(* Logix 5000 project; controller IPG_2332_07A 1769-L16ER-BB1B rev 34.12; software revision 34.01; part 2 of 4 *)
(* tags used below, declared in another part *)
   Axis_Controller : udt_Zaber_Axis;
   p_ALMD_00 : ALARM_DIGITAL;
   p_ALMD_01 : ALARM_DIGITAL;
   p_ALMD_02 : ALARM_DIGITAL;
   p_ALMD_03 : ALARM_DIGITAL;
   p_ALMD_04 : ALARM_DIGITAL;
   p_ALMD_05 : ALARM_DIGITAL;
   p_AOI_PLC_Status : AOI_PLC_Status;
   p_BarcodeDone : BOOL;
   p_CassetteGripper_Ext_IN : BOOL;
   p_CassetteGripper_OUT : BOOL;
   p_CassetteGripper_Ret_IN : BOOL;
   p_CassettePresence_IN : BOOL;
   p_CassetteRelease_IN : BOOL;   // Foot Switch
   p_Control : udt_Machine_Control_V2;   // Main Control
   p_DispenseStart_OUT : BOOL;
   p_DoorMonitor_IN : BOOL;
   p_EstopMonitor_IN : BOOL;
   p_EStopPB_IN : BOOL;
   p_EstopReset_OUT : BOOL;
   p_FerruleGripper_IN : BOOL;
   p_FerruleGripper_OUT : BOOL;
   p_FiberAxis : udt_Zaber_Axis;
   p_FiberAxis_FindPos : udt_Station_Sequence;
   p_FiberGripper_IN : BOOL;
   p_FiberGripper_OUT : BOOL;
   p_HMI_IO_Display : udt_HMI_IO_Desc;
   p_HMI_Message_Active : udt_HMI_Message_Display;
   p_HMI_Message_Sequence_Active : udt_HMI_Message_Display;
   p_HMI_PLC_Status : udt_Controller_Status;
   p_LED_01 : udt_LED;
   p_LED_02 : udt_LED;
   p_LED_03 : udt_LED;
   p_LED_04 : udt_LED;
   p_LED_Ramp_Done : BOOL;
   p_Machine_Control : udt_Machine_Control_V2;
   p_MainAirOkay_IN : BOOL;
   p_MirrorAxis : udt_Zaber_Axis;
   p_OkayToProcess : BOOL;
   p_PBLight_Amber_OUT : BOOL;
   p_PBLight_Green_OUT : BOOL;
   p_PBLight_Red_OUT : BOOL;
   p_Sequence : udt_Station_Sequence;
   p_StackLight_Amber_OUT : BOOL;
   p_StackLight_Green_OUT : BOOL;
   p_StackLight_Red_OUT : BOOL;
   p_StartPB_IN : BOOL;
   p_SyringeAxis : udt_Zaber_Axis;
   p_test_Mode : BOOL;
   p_Waiting : BOOL;
   p_WorkLight_OUT : BOOL;
   DateTime : DateTime;
   Debug_SDF : DINT;
   HMI_IO_Description : udt_IO_Desc[96];
   HMI_Messages : udt_HMI_Message_Display[48];
   HMI_Messages_Sequence : udt_HMI_Message_Display[20];
(* MainProgram_10Ms, continued *)

ROUTINE C_Alarm   (* ladder *)
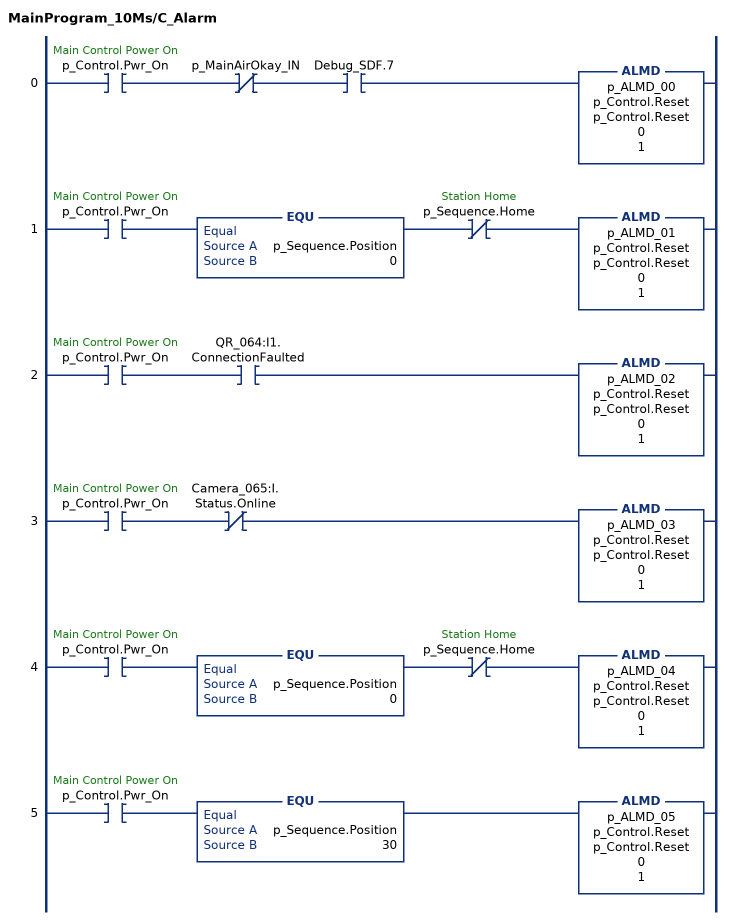
   0: XIC(p_Control.Pwr_On)XIO(p_MainAirOkay_IN)XIC(Debug_SDF.7)ALMD(p_ALMD_00,p_Control.Reset,p_Control.Reset,0,1);
   1: XIC(p_Control.Pwr_On)EQU(p_Sequence.Position,0)XIO(p_Sequence.Home)ALMD(p_ALMD_01,p_Control.Reset,p_Control.Reset,0,1);
   2: XIC(p_Control.Pwr_On)XIC(QR_064:I1.ConnectionFaulted)ALMD(p_ALMD_02,p_Control.Reset,p_Control.Reset,0,1);
   3: XIC(p_Control.Pwr_On)XIO(Camera_065:I.Status.Online)ALMD(p_ALMD_03,p_Control.Reset,p_Control.Reset,0,1);
   4: XIC(p_Control.Pwr_On)EQU(p_Sequence.Position,0)XIO(p_Sequence.Home)ALMD(p_ALMD_04,p_Control.Reset,p_Control.Reset,0,1);
   5: XIC(p_Control.Pwr_On)EQU(p_Sequence.Position,30)ALMD(p_ALMD_05,p_Control.Reset,p_Control.Reset,0,1);
END_ROUTINE

ROUTINE D_InputMapping   (* ladder *)
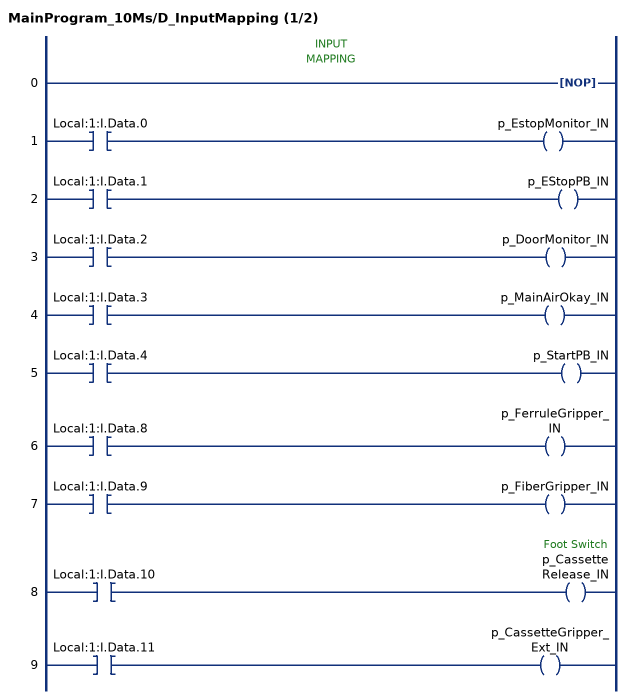
   // INPUT
   // MAPPING
   0: NOP();
   1: XIC(Local:1:I.Data.0)OTE(p_EstopMonitor_IN);
   2: XIC(Local:1:I.Data.1)OTE(p_EStopPB_IN);
   3: XIC(Local:1:I.Data.2)OTE(p_DoorMonitor_IN);
   4: XIC(Local:1:I.Data.3)OTE(p_MainAirOkay_IN);
   5: XIC(Local:1:I.Data.4)OTE(p_StartPB_IN);
   6: XIC(Local:1:I.Data.8)OTE(p_FerruleGripper_IN);
   7: XIC(Local:1:I.Data.9)OTE(p_FiberGripper_IN);
   8: XIC(Local:1:I.Data.10)OTE(p_CassetteRelease_IN);
   9: XIC(Local:1:I.Data.11)OTE(p_CassetteGripper_Ext_IN);
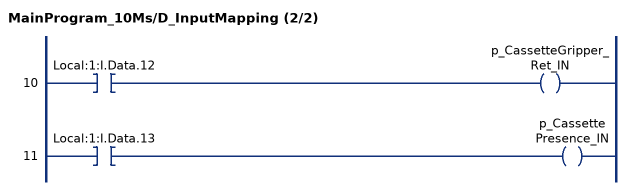
   10: XIC(Local:1:I.Data.12)OTE(p_CassetteGripper_Ret_IN);
   11: XIC(Local:1:I.Data.13)OTE(p_CassettePresence_IN);
END_ROUTINE

ROUTINE E_OutputMapping   (* ladder *)
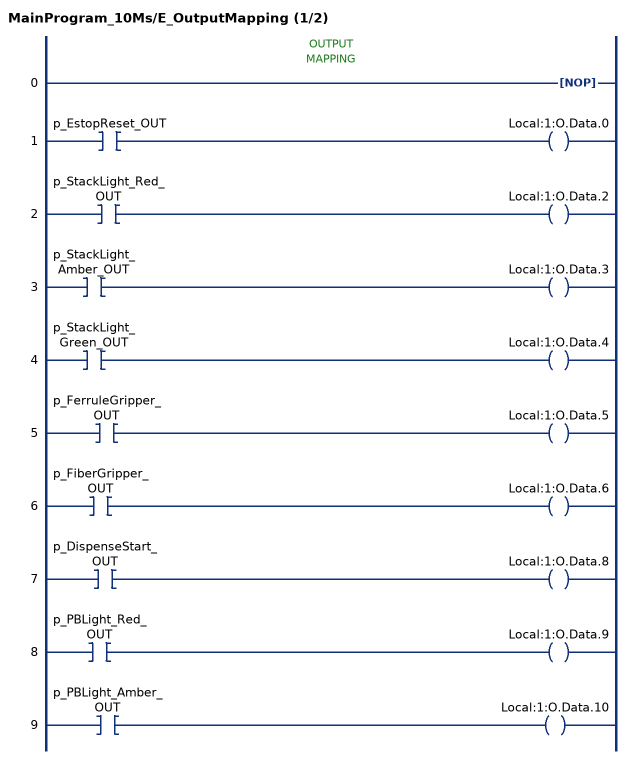
   // OUTPUT
   // MAPPING
   0: NOP();
   1: XIC(p_EstopReset_OUT)OTE(Local:1:O.Data.0);
   2: XIC(p_StackLight_Red_OUT)OTE(Local:1:O.Data.2);
   3: XIC(p_StackLight_Amber_OUT)OTE(Local:1:O.Data.3);
   4: XIC(p_StackLight_Green_OUT)OTE(Local:1:O.Data.4);
   5: XIC(p_FerruleGripper_OUT)OTE(Local:1:O.Data.5);
   6: XIC(p_FiberGripper_OUT)OTE(Local:1:O.Data.6);
   7: XIC(p_DispenseStart_OUT)OTE(Local:1:O.Data.8);
   8: XIC(p_PBLight_Red_OUT)OTE(Local:1:O.Data.9);
   9: XIC(p_PBLight_Amber_OUT)OTE(Local:1:O.Data.10);
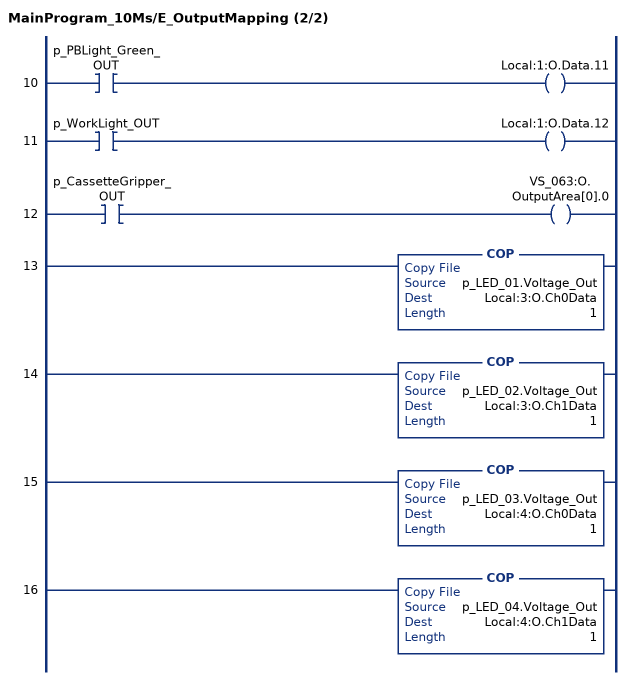
   10: XIC(p_PBLight_Green_OUT)OTE(Local:1:O.Data.11);
   11: XIC(p_WorkLight_OUT)OTE(Local:1:O.Data.12);
   12: XIC(p_CassetteGripper_OUT)OTE(VS_063:O.OutputArea[0].0);
   13: COP(p_LED_01.Voltage_Out,Local:3:O.Ch0Data,1);
   14: COP(p_LED_02.Voltage_Out,Local:3:O.Ch1Data,1);
   15: COP(p_LED_03.Voltage_Out,Local:4:O.Ch0Data,1);
   16: COP(p_LED_04.Voltage_Out,Local:4:O.Ch1Data,1);
END_ROUTINE

ROUTINE F01_HMI   (* ladder *)
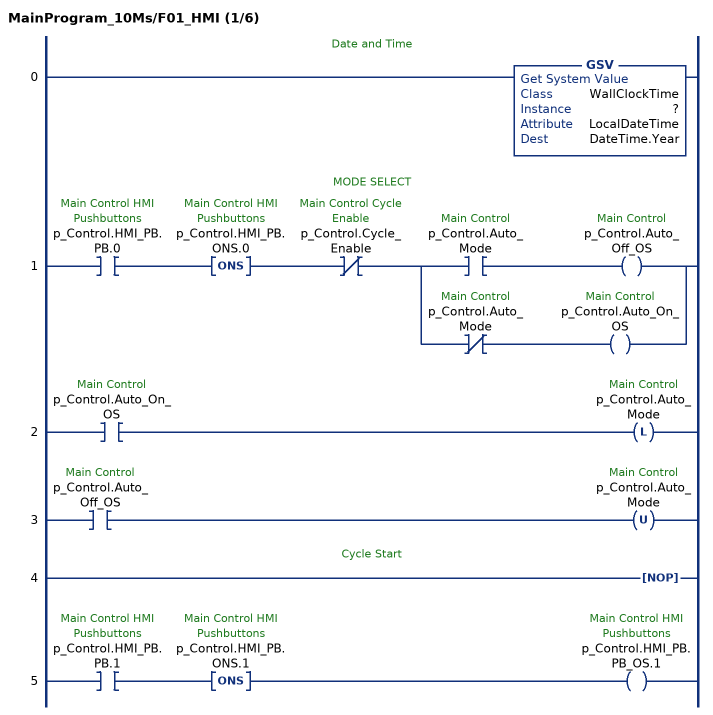
   // Date and Time
   0: GSV(WallClockTime,?,LocalDateTime,DateTime.Year);
   // MODE SELECT
   1: XIC(p_Control.HMI_PB.PB.0)ONS(p_Control.HMI_PB.ONS.0)XIO(p_Control.Cycle_Enable)[XIC(p_Control.Auto_Mode) OTE(p_Control.Auto_Off_OS) ,XIO(p_Control.Auto_Mode) OTE(p_Control.Auto_On_OS) ];
   2: XIC(p_Control.Auto_On_OS)OTL(p_Control.Auto_Mode);
   3: XIC(p_Control.Auto_Off_OS)OTU(p_Control.Auto_Mode);
   // Cycle Start
   4: NOP();
   5: XIC(p_Control.HMI_PB.PB.1)ONS(p_Control.HMI_PB.ONS.1)OTE(p_Control.HMI_PB.PB_OS.1);
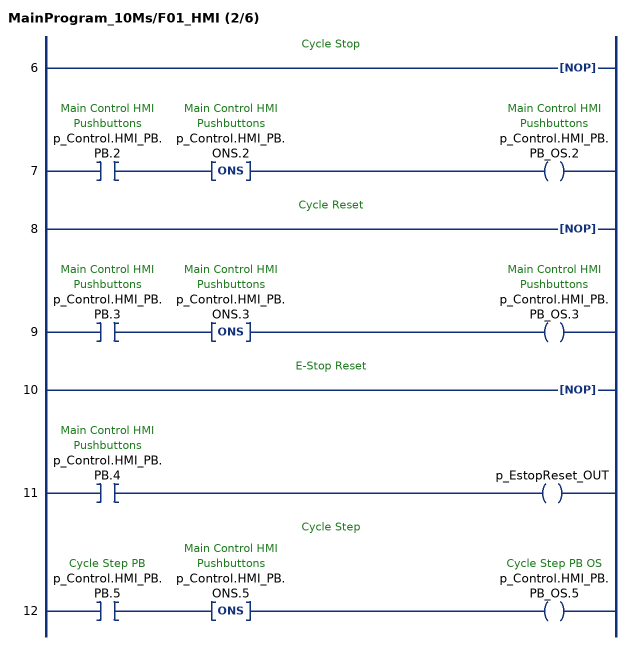
   // Cycle Stop
   6: NOP();
   7: XIC(p_Control.HMI_PB.PB.2)ONS(p_Control.HMI_PB.ONS.2)OTE(p_Control.HMI_PB.PB_OS.2);
   // Cycle Reset
   8: NOP();
   9: XIC(p_Control.HMI_PB.PB.3)ONS(p_Control.HMI_PB.ONS.3)OTE(p_Control.HMI_PB.PB_OS.3);
   // E-Stop Reset
   10: NOP();
   11: XIC(p_Control.HMI_PB.PB.4)OTE(p_EstopReset_OUT);
   // Cycle Step
   12: XIC(p_Control.HMI_PB.PB.5)ONS(p_Control.HMI_PB.ONS.5)OTE(p_Control.HMI_PB.PB_OS.5);
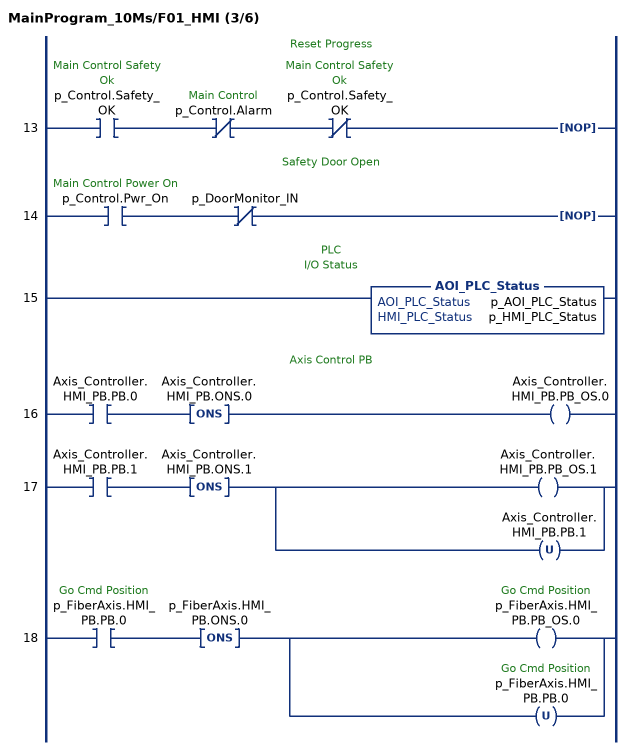
   // Reset Progress
   13: XIC(p_Control.Safety_OK)XIO(p_Control.Alarm)XIO(p_Control.Safety_OK)NOP();
   // Safety Door Open
   14: XIC(p_Control.Pwr_On)XIO(p_DoorMonitor_IN)NOP();
   // PLC
   // I/O Status
   15: AOI_PLC_Status(p_AOI_PLC_Status,p_HMI_PLC_Status);
   // Axis Control PB
   16: XIC(Axis_Controller.HMI_PB.PB.0)ONS(Axis_Controller.HMI_PB.ONS.0)OTE(Axis_Controller.HMI_PB.PB_OS.0);
   17: XIC(Axis_Controller.HMI_PB.PB.1)ONS(Axis_Controller.HMI_PB.ONS.1)[OTE(Axis_Controller.HMI_PB.PB_OS.1) ,OTU(Axis_Controller.HMI_PB.PB.1) ];
   18: XIC(p_FiberAxis.HMI_PB.PB.0)ONS(p_FiberAxis.HMI_PB.ONS.0)[OTE(p_FiberAxis.HMI_PB.PB_OS.0) ,OTU(p_FiberAxis.HMI_PB.PB.0) ];
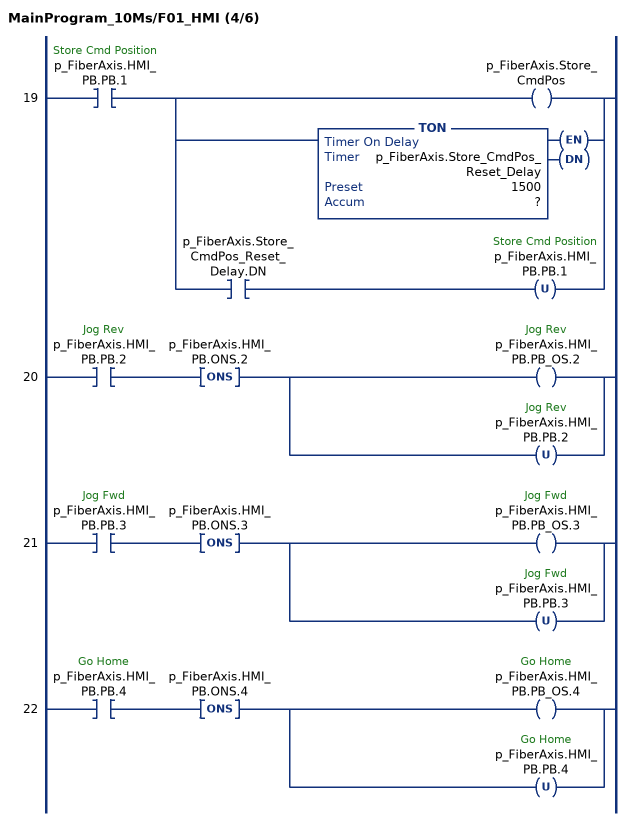
   19: XIC(p_FiberAxis.HMI_PB.PB.1)[OTE(p_FiberAxis.Store_CmdPos) ,TON(p_FiberAxis.Store_CmdPos_Reset_Delay,?,?) ,XIC(p_FiberAxis.Store_CmdPos_Reset_Delay.DN) OTU(p_FiberAxis.HMI_PB.PB.1) ];
   20: XIC(p_FiberAxis.HMI_PB.PB.2)ONS(p_FiberAxis.HMI_PB.ONS.2)[OTE(p_FiberAxis.HMI_PB.PB_OS.2) ,OTU(p_FiberAxis.HMI_PB.PB.2) ];
   21: XIC(p_FiberAxis.HMI_PB.PB.3)ONS(p_FiberAxis.HMI_PB.ONS.3)[OTE(p_FiberAxis.HMI_PB.PB_OS.3) ,OTU(p_FiberAxis.HMI_PB.PB.3) ];
   22: XIC(p_FiberAxis.HMI_PB.PB.4)ONS(p_FiberAxis.HMI_PB.ONS.4)[OTE(p_FiberAxis.HMI_PB.PB_OS.4) ,OTU(p_FiberAxis.HMI_PB.PB.4) ];
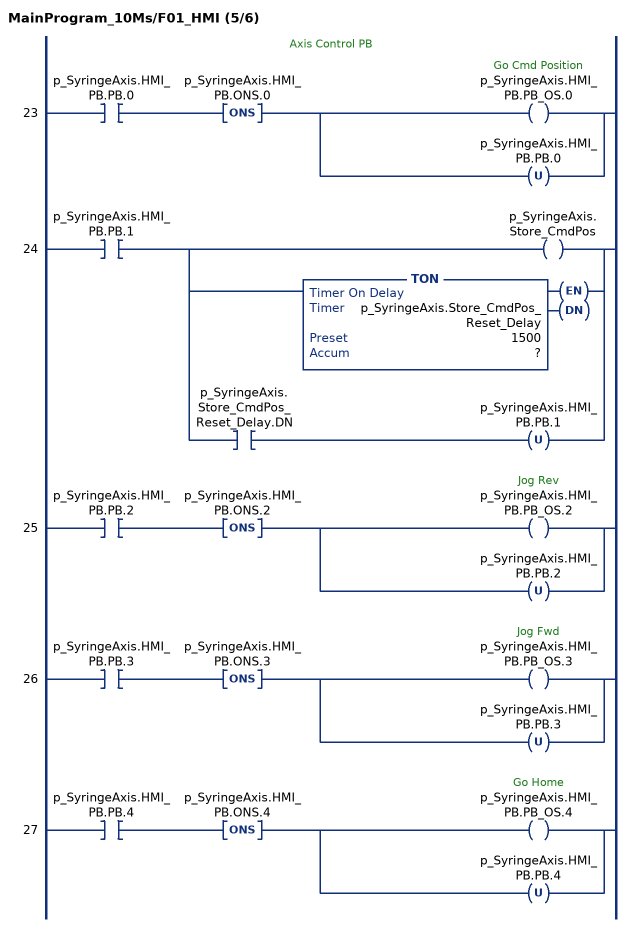
   // Axis Control PB
   23: XIC(p_SyringeAxis.HMI_PB.PB.0)ONS(p_SyringeAxis.HMI_PB.ONS.0)[OTE(p_SyringeAxis.HMI_PB.PB_OS.0) ,OTU(p_SyringeAxis.HMI_PB.PB.0) ];
   24: XIC(p_SyringeAxis.HMI_PB.PB.1)[OTE(p_SyringeAxis.Store_CmdPos) ,TON(p_SyringeAxis.Store_CmdPos_Reset_Delay,?,?) ,XIC(p_SyringeAxis.Store_CmdPos_Reset_Delay.DN) OTU(p_SyringeAxis.HMI_PB.PB.1) ];
   25: XIC(p_SyringeAxis.HMI_PB.PB.2)ONS(p_SyringeAxis.HMI_PB.ONS.2)[OTE(p_SyringeAxis.HMI_PB.PB_OS.2) ,OTU(p_SyringeAxis.HMI_PB.PB.2) ];
   26: XIC(p_SyringeAxis.HMI_PB.PB.3)ONS(p_SyringeAxis.HMI_PB.ONS.3)[OTE(p_SyringeAxis.HMI_PB.PB_OS.3) ,OTU(p_SyringeAxis.HMI_PB.PB.3) ];
   27: XIC(p_SyringeAxis.HMI_PB.PB.4)ONS(p_SyringeAxis.HMI_PB.ONS.4)[OTE(p_SyringeAxis.HMI_PB.PB_OS.4) ,OTU(p_SyringeAxis.HMI_PB.PB.4) ];
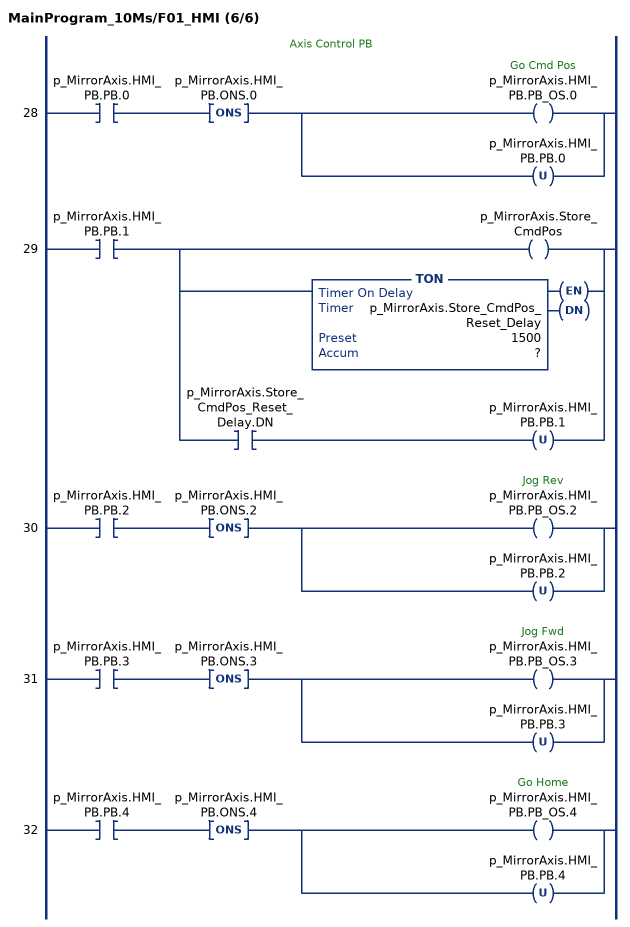
   // Axis Control PB
   28: XIC(p_MirrorAxis.HMI_PB.PB.0)ONS(p_MirrorAxis.HMI_PB.ONS.0)[OTE(p_MirrorAxis.HMI_PB.PB_OS.0) ,OTU(p_MirrorAxis.HMI_PB.PB.0) ];
   29: XIC(p_MirrorAxis.HMI_PB.PB.1)[OTE(p_MirrorAxis.Store_CmdPos) ,TON(p_MirrorAxis.Store_CmdPos_Reset_Delay,?,?) ,XIC(p_MirrorAxis.Store_CmdPos_Reset_Delay.DN) OTU(p_MirrorAxis.HMI_PB.PB.1) ];
   30: XIC(p_MirrorAxis.HMI_PB.PB.2)ONS(p_MirrorAxis.HMI_PB.ONS.2)[OTE(p_MirrorAxis.HMI_PB.PB_OS.2) ,OTU(p_MirrorAxis.HMI_PB.PB.2) ];
   31: XIC(p_MirrorAxis.HMI_PB.PB.3)ONS(p_MirrorAxis.HMI_PB.ONS.3)[OTE(p_MirrorAxis.HMI_PB.PB_OS.3) ,OTU(p_MirrorAxis.HMI_PB.PB.3) ];
   32: XIC(p_MirrorAxis.HMI_PB.PB.4)ONS(p_MirrorAxis.HMI_PB.ONS.4)[OTE(p_MirrorAxis.HMI_PB.PB_OS.4) ,OTU(p_MirrorAxis.HMI_PB.PB.4) ];
END_ROUTINE

ROUTINE F02_HMI_IO   (* ladder *)
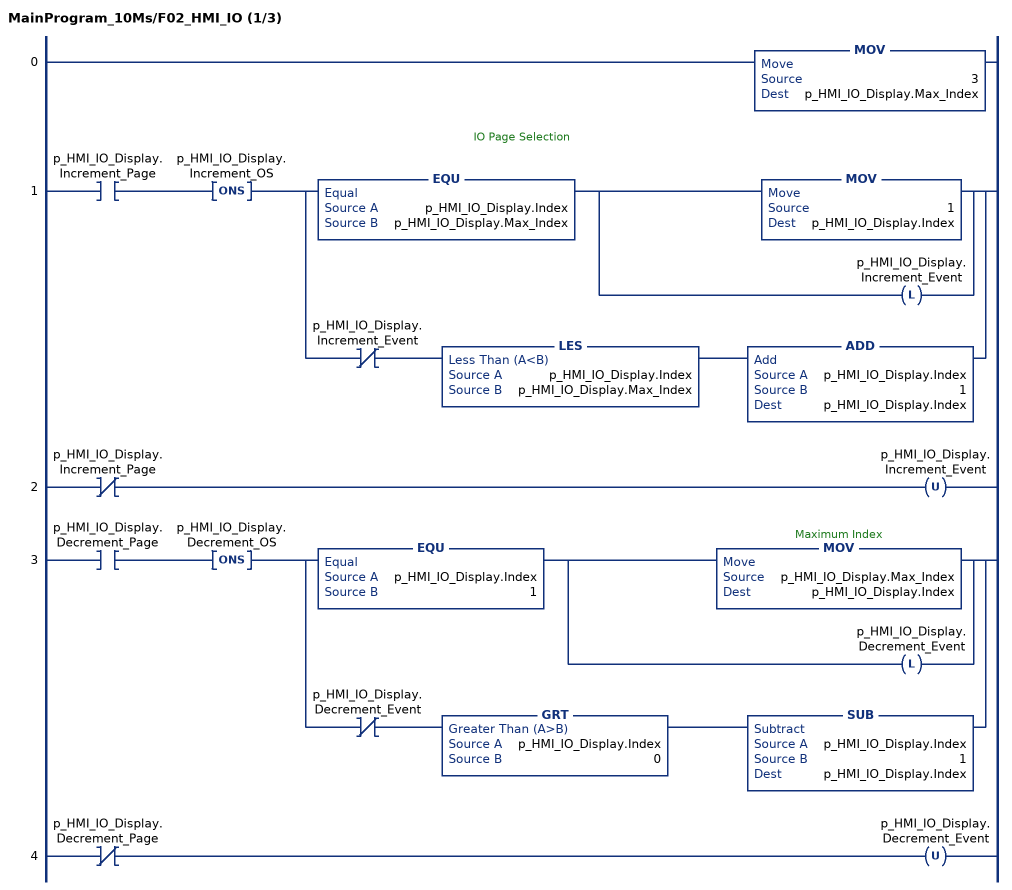
   0: MOV(3,p_HMI_IO_Display.Max_Index);
   // IO Page Selection
   1: XIC(p_HMI_IO_Display.Increment_Page)ONS(p_HMI_IO_Display.Increment_OS)[EQU(p_HMI_IO_Display.Index,p_HMI_IO_Display.Max_Index) [MOV(1,p_HMI_IO_Display.Index) ,OTL(p_HMI_IO_Display.Increment_Event) ] ,XIO(p_HMI_IO_Display.Increment_Event) LES(p_HMI_IO_Display.Index,p_HMI_IO_Display.Max_Index) ADD(p_HMI_IO_Display.Index,1,p_HMI_IO_Display.Index) ];
   2: XIO(p_HMI_IO_Display.Increment_Page)OTU(p_HMI_IO_Display.Increment_Event);
   3: XIC(p_HMI_IO_Display.Decrement_Page)ONS(p_HMI_IO_Display.Decrement_OS)[EQU(p_HMI_IO_Display.Index,1) [MOV(p_HMI_IO_Display.Max_Index,p_HMI_IO_Display.Index) ,OTL(p_HMI_IO_Display.Decrement_Event) ] ,XIO(p_HMI_IO_Display.Decrement_Event) GRT(p_HMI_IO_Display.Index,0) SUB(p_HMI_IO_Display.Index,1,p_HMI_IO_Display.Index) ];
   4: XIO(p_HMI_IO_Display.Decrement_Page)OTU(p_HMI_IO_Display.Decrement_Event);
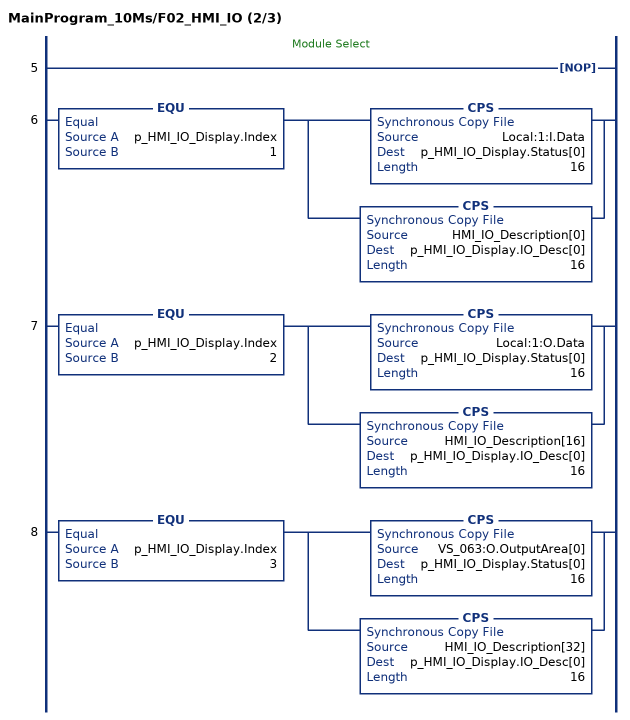
   // Module Select
   5: NOP();
   6: EQU(p_HMI_IO_Display.Index,1)[CPS(Local:1:I.Data,p_HMI_IO_Display.Status[0],16) ,CPS(HMI_IO_Description[0],p_HMI_IO_Display.IO_Desc[0],16) ];
   7: EQU(p_HMI_IO_Display.Index,2)[CPS(Local:1:O.Data,p_HMI_IO_Display.Status[0],16) ,CPS(HMI_IO_Description[16],p_HMI_IO_Display.IO_Desc[0],16) ];
   8: EQU(p_HMI_IO_Display.Index,3)[CPS(VS_063:O.OutputArea[0],p_HMI_IO_Display.Status[0],16) ,CPS(HMI_IO_Description[32],p_HMI_IO_Display.IO_Desc[0],16) ];
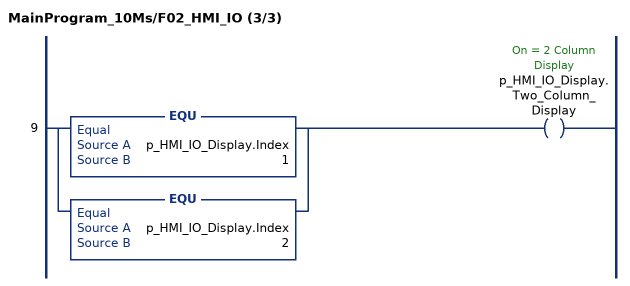
   9: [EQU(p_HMI_IO_Display.Index,1) ,EQU(p_HMI_IO_Display.Index,2) ]OTE(p_HMI_IO_Display.Two_Column_Display);
END_ROUTINE

ROUTINE F03_HMI_Messages   (* ladder *)
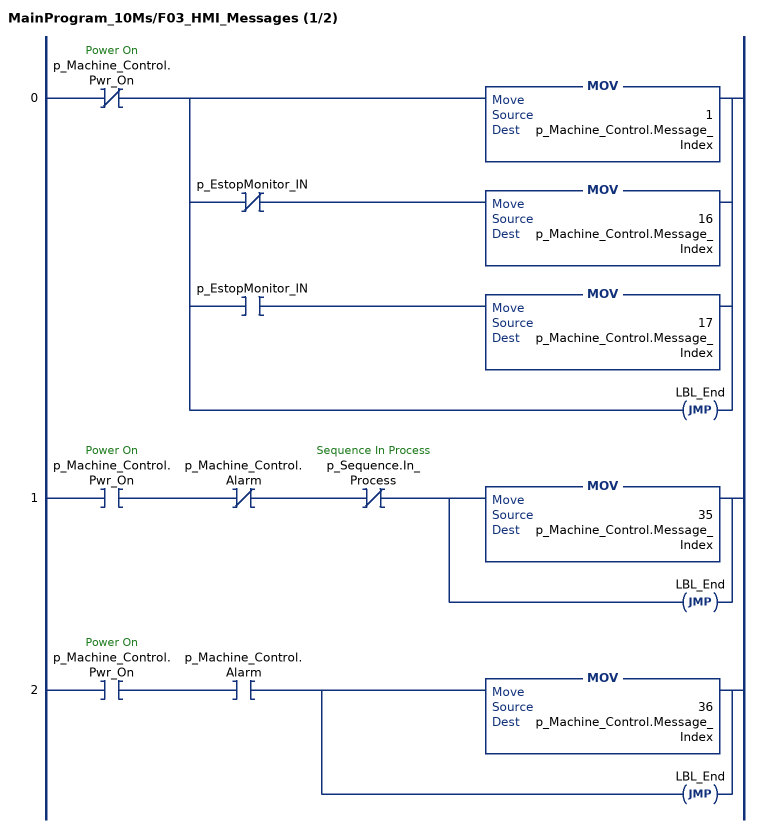
   0: XIO(p_Machine_Control.Pwr_On)[MOV(1,p_Machine_Control.Message_Index) ,XIO(p_EstopMonitor_IN) MOV(16,p_Machine_Control.Message_Index) ,XIC(p_EstopMonitor_IN) MOV(17,p_Machine_Control.Message_Index) ,JMP(LBL_End) ];
   1: XIC(p_Machine_Control.Pwr_On)XIO(p_Machine_Control.Alarm)XIO(p_Sequence.In_Process)[MOV(35,p_Machine_Control.Message_Index) ,JMP(LBL_End) ];
   2: XIC(p_Machine_Control.Pwr_On)XIC(p_Machine_Control.Alarm)[MOV(36,p_Machine_Control.Message_Index) ,JMP(LBL_End) ];
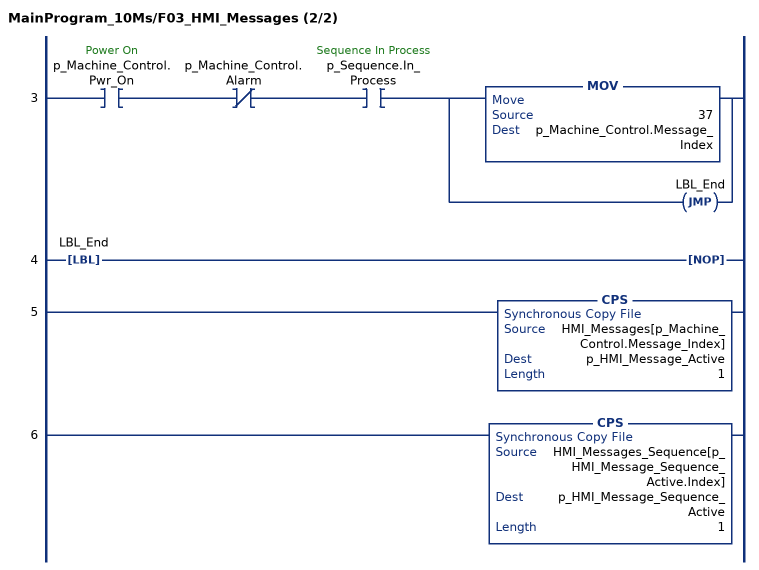
   3: XIC(p_Machine_Control.Pwr_On)XIO(p_Machine_Control.Alarm)XIC(p_Sequence.In_Process)[MOV(37,p_Machine_Control.Message_Index) ,JMP(LBL_End) ];
   4: LBL(LBL_End)NOP();
   5: CPS(HMI_Messages[p_Machine_Control.Message_Index],p_HMI_Message_Active,1);
   6: CPS(HMI_Messages_Sequence[p_HMI_Message_Sequence_Active.Index],p_HMI_Message_Sequence_Active,1);
END_ROUTINE

ROUTINE G_Sequence   (* ladder *)
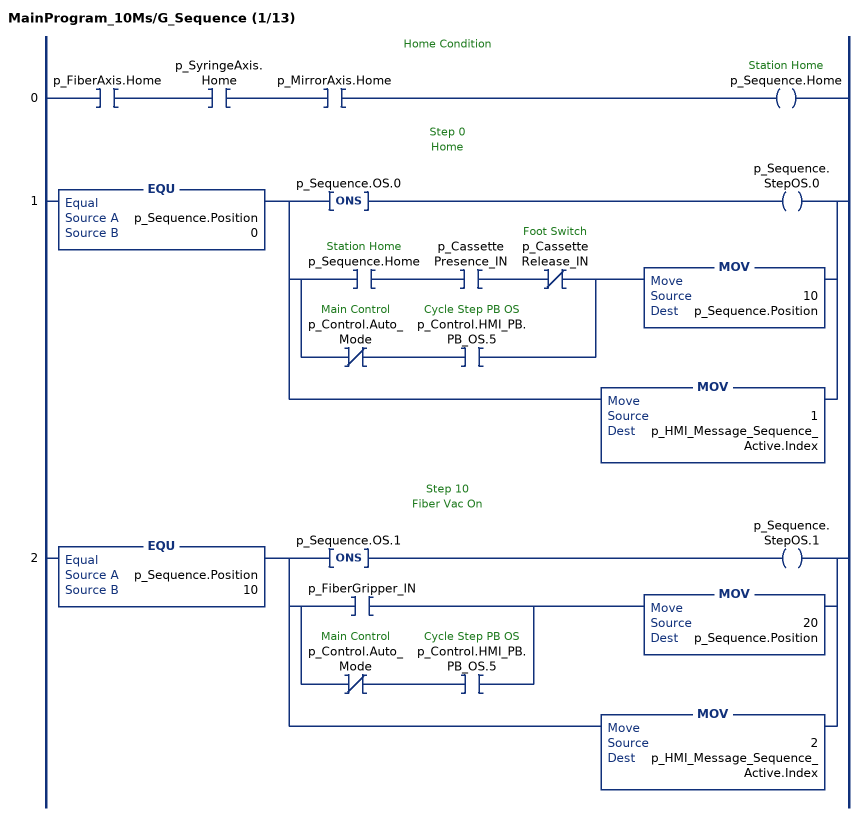
   // Home Condition
   0: XIC(p_FiberAxis.Home)XIC(p_SyringeAxis.Home)XIC(p_MirrorAxis.Home)OTE(p_Sequence.Home);
   // Step 0
   // Home
   1: EQU(p_Sequence.Position,0)[ONS(p_Sequence.OS.0) OTE(p_Sequence.StepOS.0) ,[XIC(p_Sequence.Home) XIC(p_CassettePresence_IN) XIO(p_CassetteRelease_IN) ,XIO(p_Control.Auto_Mode) XIC(p_Control.HMI_PB.PB_OS.5) ] MOV(10,p_Sequence.Position) ,MOV(1,p_HMI_Message_Sequence_Active.Index) ];
   // Step 10
   // Fiber Vac On
   2: EQU(p_Sequence.Position,10)[ONS(p_Sequence.OS.1) OTE(p_Sequence.StepOS.1) ,[XIC(p_FiberGripper_IN) ,XIO(p_Control.Auto_Mode) XIC(p_Control.HMI_PB.PB_OS.5) ] MOV(20,p_Sequence.Position) ,MOV(2,p_HMI_Message_Sequence_Active.Index) ];
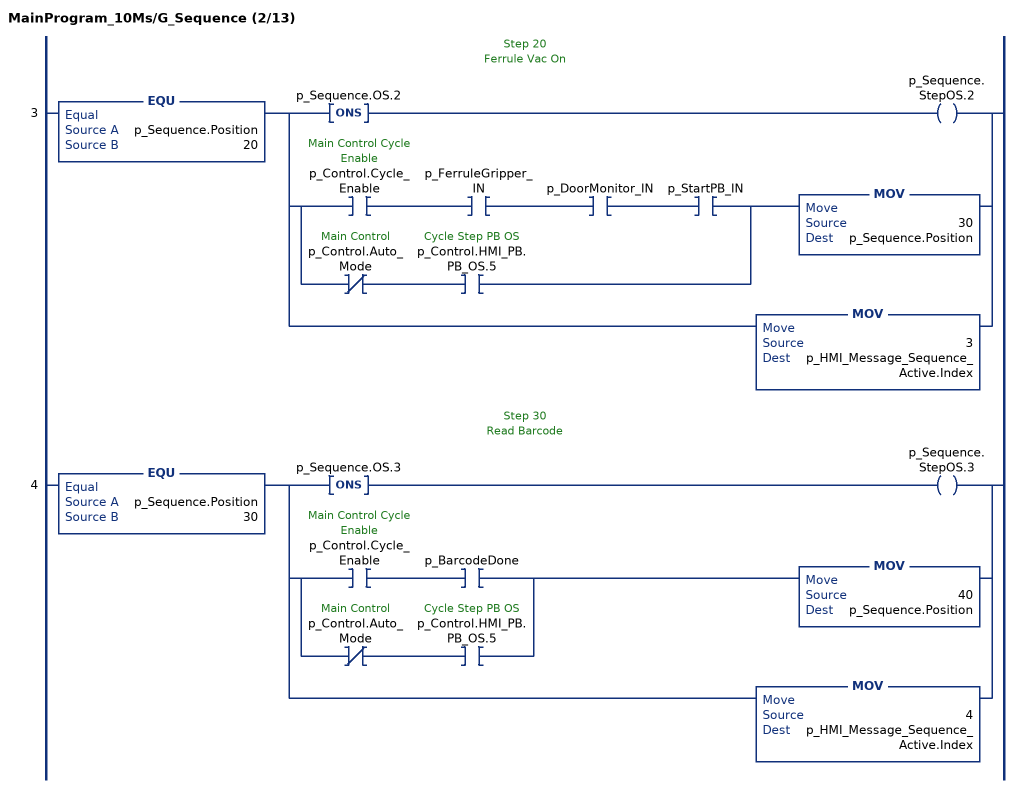
   // Step 20
   // Ferrule Vac On
   3: EQU(p_Sequence.Position,20)[ONS(p_Sequence.OS.2) OTE(p_Sequence.StepOS.2) ,[XIC(p_Control.Cycle_Enable) XIC(p_FerruleGripper_IN) XIC(p_DoorMonitor_IN) XIC(p_StartPB_IN) ,XIO(p_Control.Auto_Mode) XIC(p_Control.HMI_PB.PB_OS.5) ] MOV(30,p_Sequence.Position) ,MOV(3,p_HMI_Message_Sequence_Active.Index) ];
   // Step 30
   // Read Barcode
   4: EQU(p_Sequence.Position,30)[ONS(p_Sequence.OS.3) OTE(p_Sequence.StepOS.3) ,[XIC(p_Control.Cycle_Enable) XIC(p_BarcodeDone) ,XIO(p_Control.Auto_Mode) XIC(p_Control.HMI_PB.PB_OS.5) ] MOV(40,p_Sequence.Position) ,MOV(4,p_HMI_Message_Sequence_Active.Index) ];
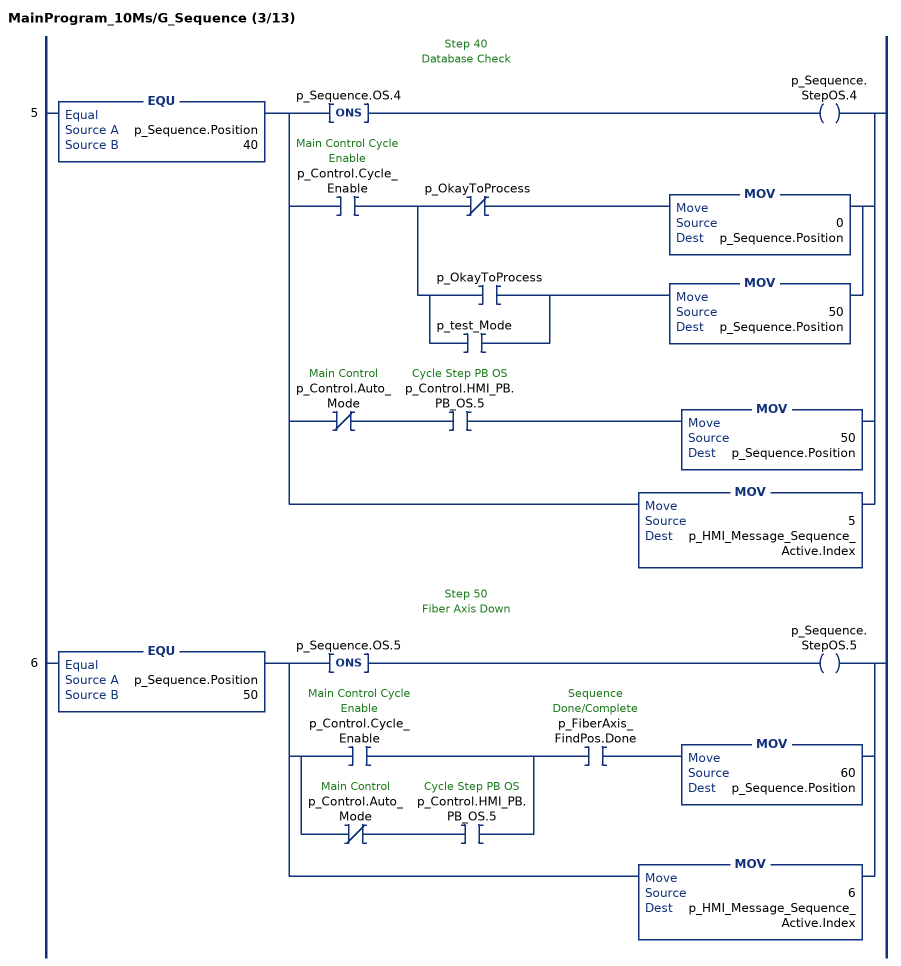
   // Step 40
   // Database Check
   5: EQU(p_Sequence.Position,40)[ONS(p_Sequence.OS.4) OTE(p_Sequence.StepOS.4) ,XIC(p_Control.Cycle_Enable) [XIO(p_OkayToProcess) MOV(0,p_Sequence.Position) ,[XIC(p_OkayToProcess) ,XIC(p_test_Mode) ] MOV(50,p_Sequence.Position) ] ,XIO(p_Control.Auto_Mode) XIC(p_Control.HMI_PB.PB_OS.5) MOV(50,p_Sequence.Position) ,MOV(5,p_HMI_Message_Sequence_Active.Index) ];
   // Step 50
   // Fiber Axis Down
   6: EQU(p_Sequence.Position,50)[ONS(p_Sequence.OS.5) OTE(p_Sequence.StepOS.5) ,[XIC(p_Control.Cycle_Enable) ,XIO(p_Control.Auto_Mode) XIC(p_Control.HMI_PB.PB_OS.5) ] XIC(p_FiberAxis_FindPos.Done) MOV(60,p_Sequence.Position) ,MOV(6,p_HMI_Message_Sequence_Active.Index) ];
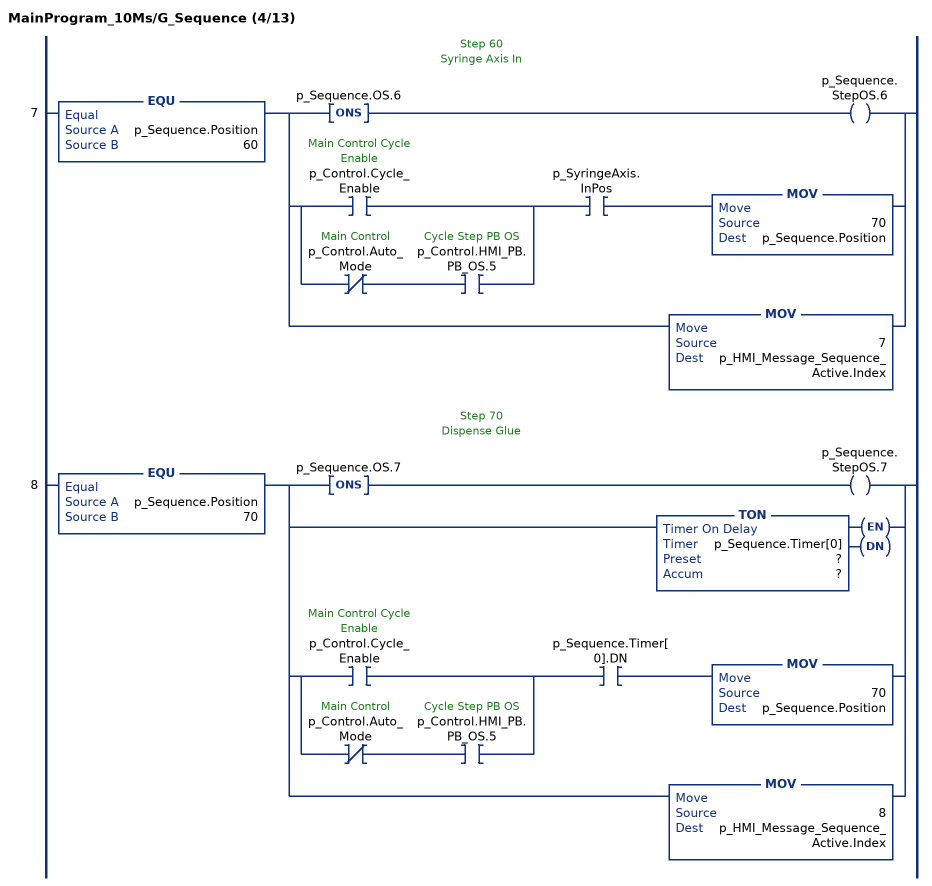
   // Step 60
   // Syringe Axis In
   7: EQU(p_Sequence.Position,60)[ONS(p_Sequence.OS.6) OTE(p_Sequence.StepOS.6) ,[XIC(p_Control.Cycle_Enable) ,XIO(p_Control.Auto_Mode) XIC(p_Control.HMI_PB.PB_OS.5) ] XIC(p_SyringeAxis.InPos) MOV(70,p_Sequence.Position) ,MOV(7,p_HMI_Message_Sequence_Active.Index) ];
   // Step 70
   // Dispense Glue
   8: EQU(p_Sequence.Position,70)[ONS(p_Sequence.OS.7) OTE(p_Sequence.StepOS.7) ,TON(p_Sequence.Timer[0],?,?) ,[XIC(p_Control.Cycle_Enable) ,XIO(p_Control.Auto_Mode) XIC(p_Control.HMI_PB.PB_OS.5) ] XIC(p_Sequence.Timer[0].DN) MOV(70,p_Sequence.Position) ,MOV(8,p_HMI_Message_Sequence_Active.Index) ];
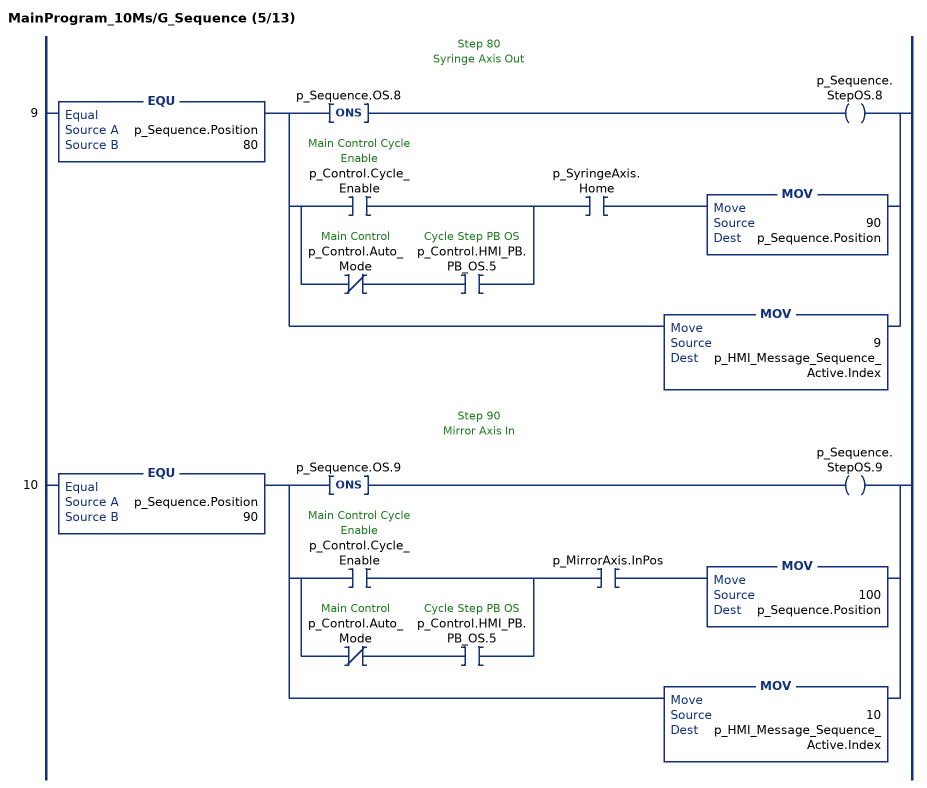
   // Step 80
   // Syringe Axis Out
   9: EQU(p_Sequence.Position,80)[ONS(p_Sequence.OS.8) OTE(p_Sequence.StepOS.8) ,[XIC(p_Control.Cycle_Enable) ,XIO(p_Control.Auto_Mode) XIC(p_Control.HMI_PB.PB_OS.5) ] XIC(p_SyringeAxis.Home) MOV(90,p_Sequence.Position) ,MOV(9,p_HMI_Message_Sequence_Active.Index) ];
   // Step 90
   // Mirror Axis In
   10: EQU(p_Sequence.Position,90)[ONS(p_Sequence.OS.9) OTE(p_Sequence.StepOS.9) ,[XIC(p_Control.Cycle_Enable) ,XIO(p_Control.Auto_Mode) XIC(p_Control.HMI_PB.PB_OS.5) ] XIC(p_MirrorAxis.InPos) MOV(100,p_Sequence.Position) ,MOV(10,p_HMI_Message_Sequence_Active.Index) ];
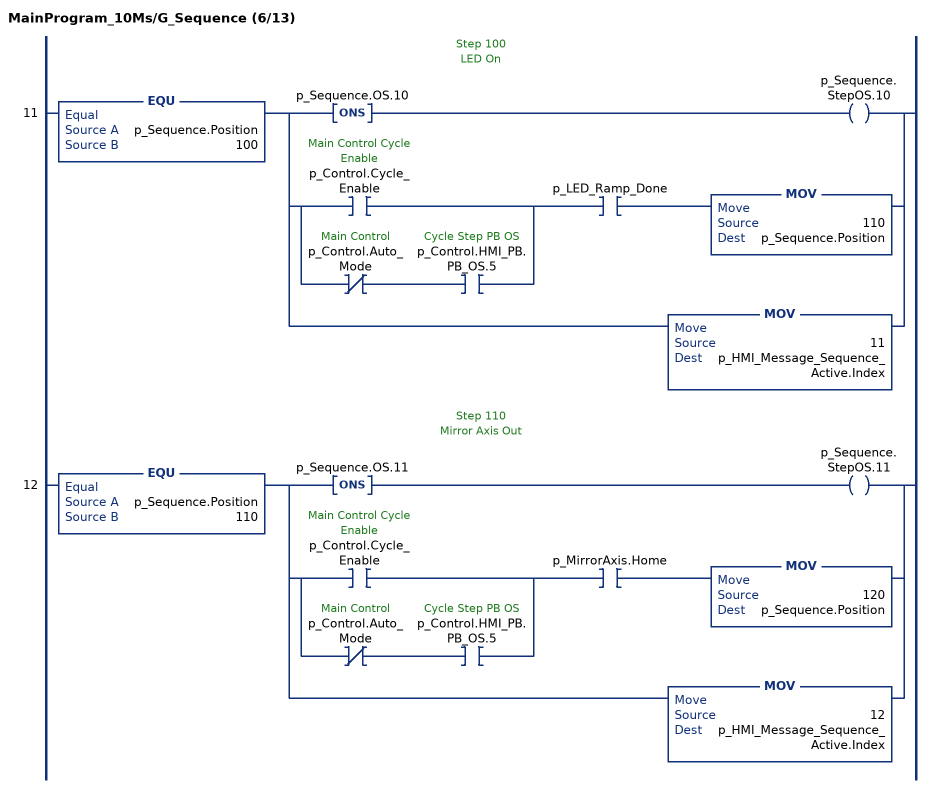
   // Step 100
   // LED On
   11: EQU(p_Sequence.Position,100)[ONS(p_Sequence.OS.10) OTE(p_Sequence.StepOS.10) ,[XIC(p_Control.Cycle_Enable) ,XIO(p_Control.Auto_Mode) XIC(p_Control.HMI_PB.PB_OS.5) ] XIC(p_LED_Ramp_Done) MOV(110,p_Sequence.Position) ,MOV(11,p_HMI_Message_Sequence_Active.Index) ];
   // Step 110
   // Mirror Axis Out
   12: EQU(p_Sequence.Position,110)[ONS(p_Sequence.OS.11) OTE(p_Sequence.StepOS.11) ,[XIC(p_Control.Cycle_Enable) ,XIO(p_Control.Auto_Mode) XIC(p_Control.HMI_PB.PB_OS.5) ] XIC(p_MirrorAxis.Home) MOV(120,p_Sequence.Position) ,MOV(12,p_HMI_Message_Sequence_Active.Index) ];
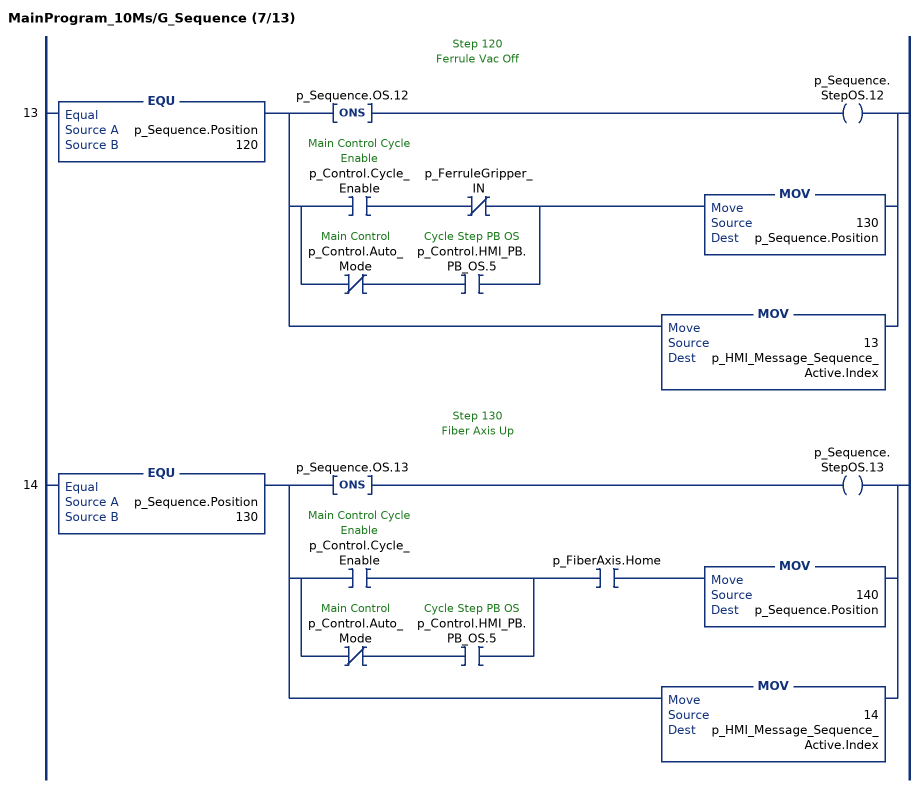
   // Step 120
   // Ferrule Vac Off
   13: EQU(p_Sequence.Position,120)[ONS(p_Sequence.OS.12) OTE(p_Sequence.StepOS.12) ,[XIC(p_Control.Cycle_Enable) XIO(p_FerruleGripper_IN) ,XIO(p_Control.Auto_Mode) XIC(p_Control.HMI_PB.PB_OS.5) ] MOV(130,p_Sequence.Position) ,MOV(13,p_HMI_Message_Sequence_Active.Index) ];
   // Step 130
   // Fiber Axis Up
   14: EQU(p_Sequence.Position,130)[ONS(p_Sequence.OS.13) OTE(p_Sequence.StepOS.13) ,[XIC(p_Control.Cycle_Enable) ,XIO(p_Control.Auto_Mode) XIC(p_Control.HMI_PB.PB_OS.5) ] XIC(p_FiberAxis.Home) MOV(140,p_Sequence.Position) ,MOV(14,p_HMI_Message_Sequence_Active.Index) ];
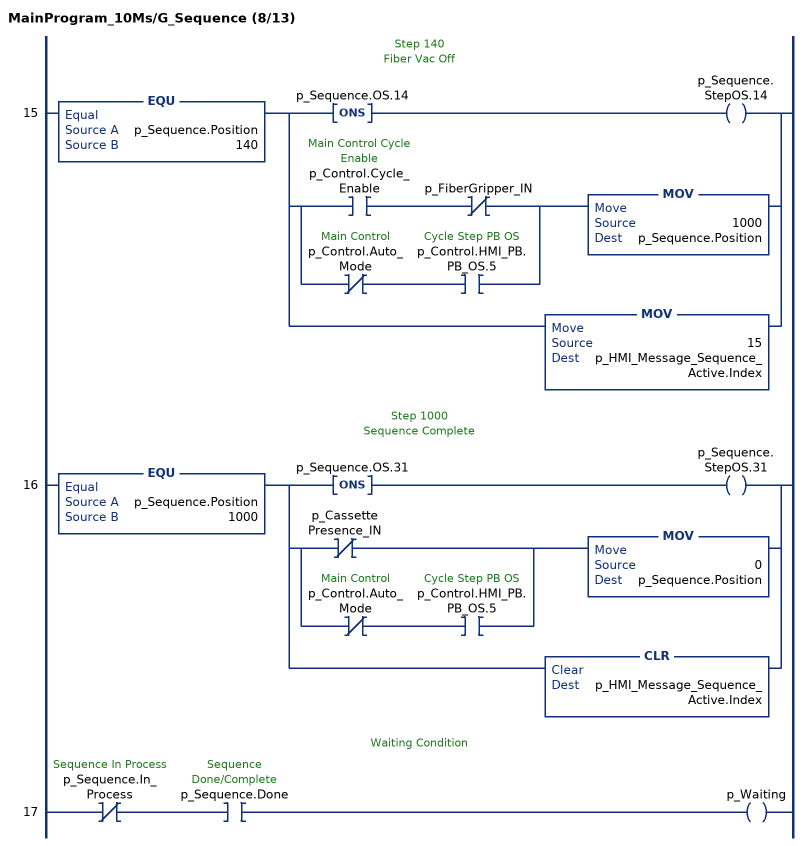
   // Step 140
   // Fiber Vac Off
   15: EQU(p_Sequence.Position,140)[ONS(p_Sequence.OS.14) OTE(p_Sequence.StepOS.14) ,[XIC(p_Control.Cycle_Enable) XIO(p_FiberGripper_IN) ,XIO(p_Control.Auto_Mode) XIC(p_Control.HMI_PB.PB_OS.5) ] MOV(1000,p_Sequence.Position) ,MOV(15,p_HMI_Message_Sequence_Active.Index) ];
   // Step 1000
   // Sequence Complete
   16: EQU(p_Sequence.Position,1000)[ONS(p_Sequence.OS.31) OTE(p_Sequence.StepOS.31) ,[XIO(p_CassettePresence_IN) ,XIO(p_Control.Auto_Mode) XIC(p_Control.HMI_PB.PB_OS.5) ] MOV(0,p_Sequence.Position) ,CLR(p_HMI_Message_Sequence_Active.Index) ];
   // Waiting Condition
   17: XIO(p_Sequence.In_Process)XIC(p_Sequence.Done)OTE(p_Waiting);
